// TwinCAT 3 PLC project OptimizationExample
// ProgramVersion: 3.1.4024.0
// libraries:
//   Tc2_Standard, * (Beckhoff Automation GmbH)
//   Tc2_System, * (Beckhoff Automation GmbH)
//   Tc2_Utilities, * (Beckhoff Automation GmbH)
//   Tc3_Module, * (Beckhoff Automation GmbH)
// project tree:
//   / PlcTask.TcTTO
//   POUs/ Interface_TcCOM.TcPOU, MAIN.TcPOU
// real-time tasks:
//   TASK PlcTask: cycle T#10ms, priority 20, ADS port 350

CONFIGURATION OptimizationExample
    RESOURCE PLC ON TwinCAT3
        TASK PlcTask(INTERVAL := T#10ms, PRIORITY := 20);
        PROGRAM MAIN WITH PlcTask : MAIN;
    END_RESOURCE
END_CONFIGURATION

// ---- POUs/MAIN.TcPOU
PROGRAM MAIN
VAR
	
	x1 : LREAL := -2;
	x2 : LREAL := 444;

	solution : ARRAY[0..7] OF LREAL;	

	fb_QPopt : Interface_TcCOM;
	
	TimeProfiler : Profiler;
END_VAR

TimeProfiler(START := TRUE, RESET := TRUE);

fb_QPopt.ip.solve(in1:= ADR(x1),  out1:= ADR(solution));

TimeProfiler(START := FALSE);

END_PROGRAM

// ---- POUs/Interface_TcCOM.TcPOU
FUNCTION_BLOCK Interface_TcCOM
// Interface to TcCOM object
//  1. define the interface pointer (ip)
//  2. define the interface ID      (iid)
VAR_OUTPUT
	ip : I_QPopt;  // (1.) C++ projekt -> .tmc -> Data Types -> InterfaceNAME
END_VAR
VAR
	{attribute 'TcInitSymbol'}
	nObjId : OTCID; 	// Instance configured to be retrieved
	iid : IID :=  TC_GLOBAL_IID_LIST.IID_I_QPopt; // (2.) TC_GLOBAL_IID_LIST.IID_InterfaceNAME;
	hrInit : HRESULT;
END_VAR

METHOD FB_exit : BOOL
VAR_INPUT
	bInCopyCode : BOOL; // if TRUE, the exit method is called for exiting an instance that is copied afterwards (online change).
END_VAR
IF NOT bInCopyCode THEN // if not online change
	FW_SafeRelease(ADR(ip));
END_IF
END_METHOD

METHOD FB_init : BOOL
VAR_INPUT
	bInitRetains : BOOL; // if TRUE, the retain variables are initialized (warm start / cold start)
	bInCopyCode : BOOL;  // if TRUE, the instance afterwards gets moved into the copy code (online change)
END_VAR
IF NOT bInCopyCode THEN // if not online change
	IF nObjID <> 0 THEN
		hrInit := FW_ObjMgr_GetObjectInstance(oid:=nObjID, iid:=iid, pipUnk:=ADR(ip));
	ELSE
		hrInit := E_HRESULTAdsErr.INVALIDOBJID;
	END_IF
END_IF
END_METHOD

END_FUNCTION_BLOCK
